// TIA Portal V21 export
TYPE "Std_Stazioni"
   STRUCT
      IN : Struct
         Possibile : Bool;
         Selezionato : Bool;
         Attivo : Bool;
      END_STRUCT;
      Prm : Struct
         PrioritaInvioProdotto : "Std_Priorità";
         PrioritaRicezioneProdotto : "Std_Priorità";
      END_STRUCT;
   END_STRUCT;
END_TYPE
